// SIMATIC S7-200 project (STEP 7-Micro/WIN), CPU 226 CN REL 02.01

SYMBOL_TABLE USER1
Sens_Tub_Inf     I0.0     // Sensor fotoelectrico del tubo inferior (nivel bajo de stock)
Sens_Tub_Sup     I0.1     // Sensor fotoelectrico del tubo superior (nivel alto de stock)
Sens_Sal_Tub     I0.2     // Sensor de presencia a la salida del tubo dosificador
Sens_Pieza_Rec   I0.3     // Sensor de presencia de pieza lista para recoger
Sens_Fibra_Pza   I0.4     // Sensor de fibra omron (pieza grande receptora presente)
CilS_Ext         I0.5     // Sensor cilindro superior extendido (sujetador OK)
CilS_Ret         I0.6     // Sensor cilindro superior retraido
CilI_Ext         I0.7     // Sensor cilindro inferior extendido
CilI_Ret         I1.0     // Sensor cilindro inferior retraido (pieza liberada)
Giro_AH          I1.1     // Sensor giro antihorario alcanzado (posicion recogida)
Giro_H           I1.2     // Sensor giro horario alcanzado (posicion origen)
Pinza_Cer        I1.3     // Sensor cierre de la pinza de agarre
CilV_Abajo       I1.4     // Sensor cilindro vertical hacia abajo
CilV_Arriba      I1.5     // Sensor cilindro vertical hacia arriba
CilH_Atras       I1.6     // Sensor cilindro horizontal hacia atras (origen)
CilH_Adelante    I1.7     // Sensor cilindro horizontal hacia adelante (sobre pieza)
Btn_Rojo         I2.4     // Boton de parada
Btn_Verde        I2.5     // Boton de marcha
Seta_Emerg       I2.6     // Seta de emergencia (NC - 0 = emergencia activa)
Selector         I2.7     // Selector rotatorio de modo
V_CilI           Q0.0     // Valvula cilindro inferior (liberador) - activa en P2
V_CilS           Q0.1     // Valvula cilindro superior (sujetador) - activa en P1 y P2
V_Giro_H         Q0.2     // Valvula cilindro rotatorio antihorario - activa en P4 a P7
V_Pinza          Q0.3     // Valvula garra (cerrar pinza) - activa en P6 a P9
V_CilV           Q0.4     // Valvula cilindro vertical (bajar) - activa en P5 P6 P9 P10
V_CilH           Q0.5     // Valvula cilindro horizontal (adelante) - activa en P8 a P11
Baliza_Roja      Q0.6     // Baliza roja - sin stock en reposo
Baliza_Amarilla  Q0.7     // Baliza amarilla - parada activa (M6.0)
Baliza_Verde     Q1.0     // Baliza verde - ciclo en ejecucion
Led_Amarillo     Q1.5     // LED boton amarillo - parada activa
Led_Verde        Q1.6     // LED boton verde - ciclo en ejecucion
Led_Rojo         Q1.7     // LED boton rojo - sin stock en reposo
P0_Reposo        M0.0     // Plaza P0 - Estado reposo (marcado inicial)
P1_Dos_Sujetar   M0.1     // Plaza P1 - Cilindro superior sujetando columna
P2_Dos_Caida     M0.2     // Plaza P2 - Cilindro inferior retraido (pieza en caida)
P3_Dos_Restaurar M0.3     // Plaza P3 - Dosificador retornando a posicion base
P4_Mesa_Giro     M0.4     // Plaza P4 - Mesa girando a posicion de recogida
P5_Pick_Bajar    M0.5     // Plaza P5 - Garra descendiendo sobre pieza secundaria
P6_Pick_Agarrar  M0.6     // Plaza P6 - Pinza cerrando para sujetar la pieza
P7_Pick_Subir    M0.7     // Plaza P7 - Garra subiendo con pieza sujeta
P8_Place_Trans   M1.0     // Plaza P8 - Brazo trasladando horizontalmente a base
P9_Place_Bajar   M1.1     // Plaza P9 - Garra bajando para insertar en base
P10_Place_Soltar M1.2     // Plaza P10 - Pinza abriendo para liberar pieza
P11_Place_Subir  M1.3     // Plaza P11 - Garra subiendo tras ensamblaje
P12_Reset_Arm    M1.4     // Plaza P12 - Retorno horizontal y mesa a origen
Ev_Marcha        M2.0     // Evento - Boton de marcha activo
Ev_Tub_Inf       M2.1     // Evento - Stock disponible en tubo (nivel bajo)
Ev_Fibra         M2.2     // Evento - Pieza grande receptora detectada
Ev_CilS_Ext      M2.3     // Evento - Cilindro superior extendido confirmado
Ev_CilS_Ret      M2.4     // Evento - Cilindro superior retraido confirmado
Ev_CilI_Ext      M2.5     // Evento - Cilindro inferior extendido confirmado
Ev_CilI_Ret      M2.6     // Evento - Cilindro inferior retraido (pieza liberada)
Ev_Giro_AH       M2.7     // Evento - Giro antihorario alcanzado (posicion recogida)
Ev_Giro_H        M3.0     // Evento - Giro horario alcanzado (posicion origen)
Ev_Pinza_Cer     M3.1     // Evento - Pinza cerrada (agarre confirmado)
Ev_CilV_Abajo    M3.2     // Evento - Cilindro vertical en posicion abajo
Ev_CilV_Arriba   M3.3     // Evento - Cilindro vertical en posicion arriba
Ev_CilH_Atras    M3.4     // Evento - Cilindro horizontal en posicion atras
Ev_CilH_Adel     M3.5     // Evento - Cilindro horizontal en posicion adelante
T0_Inicio        M4.0     // Disparo T0 - Condicion para iniciar ciclo (P0->P1)
T1_SujecOK       M4.1     // Disparo T1 - Sujecion de columna confirmada (P1->P2)
T2_PiezaCaida    M4.2     // Disparo T2 - Pieza liberada y caida (P2->P3)
T3_DosifRest     M4.3     // Disparo T3 - Dosificador restaurado (P3->P4)
T4_MesaRec       M4.4     // Disparo T4 - Mesa en posicion recogida (P4->P5)
T5_GarraAbajo    M4.5     // Disparo T5 - Garra en contacto con pieza (P5->P6)
T6_AgarreOK      M4.6     // Disparo T6 - Agarre de pieza confirmado (P6->P7)
T7_PiezaElev     M4.7     // Disparo T7 - Pieza secundaria elevada (P7->P8)
T8_BrazoAdel     M5.0     // Disparo T8 - Brazo en punto de entrega (P8->P9)
T9_PiezaBase     M5.1     // Disparo T9 - Pieza posicionada en base grande (P9->P10)
T10_PinzaAb      M5.2     // Disparo T10 - Pinza abierta pieza liberada (P10->P11)
T11_GarraRet     M5.3     // Disparo T11 - Garra retirada del ensamblaje (P11->P12)
T12_FinCiclo     M5.4     // Disparo T12 - Sistema en origen fin de ciclo (P12->P0)
Flag_Parada      M6.0     // Flag de parada - activado por flanco Btn_Rojo reset en P0
Sol_ES           V0.0     // Solicitud Ensamblaje a Seleccion
Ack_Sol_ES       V1.0     // Reconocimiento ES
Ack_ME           V0.1     // Reconocimiento marcha Unidad de Ensamblaje
Marcha_E         V1.1     // Solicitud de marcha para la Unidad de Ensamblaje
Ens_OK           V0.2     // Unidad de Ensamblaje disponible
END_SYMBOL_TABLE

SYMBOL_TABLE S7-200 Symbols
First_Scan_On    SM0.1    // 仅第一个扫描周期中接通为 ON
END_SYMBOL_TABLE

ORGANIZATION_BLOCK MAIN:OB1
TITLE=UNIDAD DE ENSAMBLAJE - RED DE PETRI CIPN v2
//  ===========================================================
//  MODULO 0: SEGURIDAD - EMERGENCIA (Evaluado primero, cada scan)
//  Si Seta = 0 (NC abierta) -> Reset total, fuerza P0, apaga salidas.
//  ===========================================================
BEGIN
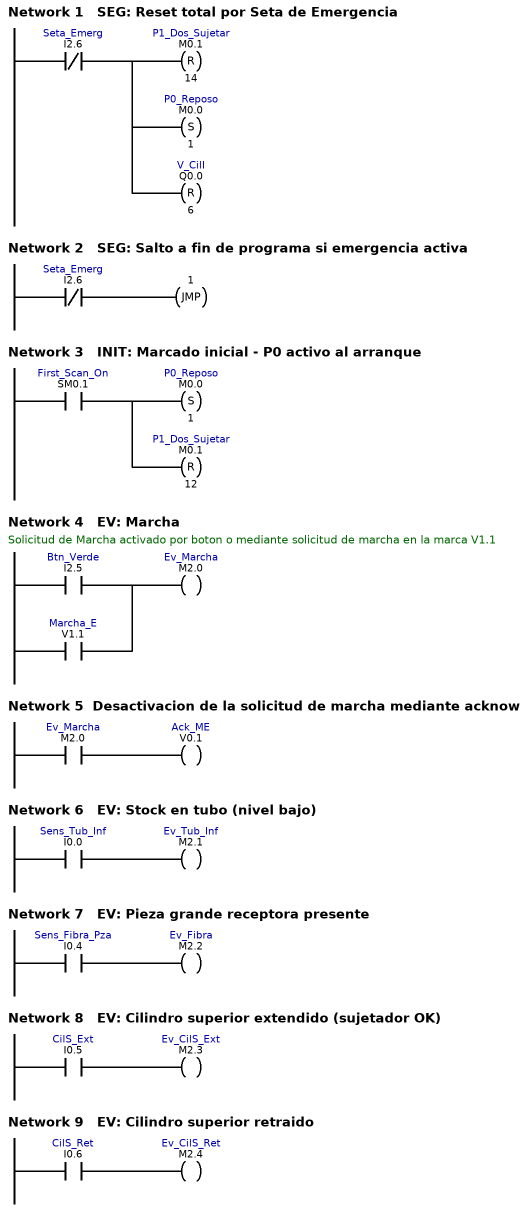
Network 1 //  SEG: Reset total por Seta de Emergencia
LDN    Seta_Emerg:I2.6
R      P1_Dos_Sujetar:M0.1, 14
S      P0_Reposo:M0.0, 1
R      V_CilI:Q0.0, 6
Network 2 //  SEG: Salto a fin de programa si emergencia activa
// ===========================================================
// MODULO 1: INICIALIZACION
// Ejecuta solo en el primer scan (SM0.1 = 1 unicamente en scan 1).
// Establece marcado inicial: P0 activo, resto limpio.
// ===========================================================
LDN    Seta_Emerg:I2.6
JMP    1
Network 3 //  INIT: Marcado inicial - P0 activo al arranque
// ===========================================================
// MODULO 2: EVENTOS (CAPTURA DE SENSORES)
// Copia directa de entradas a marcas de evento para desacoplar
// la logica secuencial de las senales fisicas.
// ===========================================================
LD     First_Scan_On:SM0.1
S      P0_Reposo:M0.0, 1
R      P1_Dos_Sujetar:M0.1, 12
Network 4 //  EV: Marcha 
//  Solicitud de Marcha activado por boton o mediante solicitud de marcha en la marca V1.1
LD     Btn_Verde:I2.5
O      Marcha_E:V1.1
=      Ev_Marcha:M2.0
Network 5 // Desactivacion de la solicitud de marcha mediante acknowledgement
LD     Ev_Marcha:M2.0
=      Ack_ME:V0.1
Network 6 //  EV: Stock en tubo (nivel bajo)
LD     Sens_Tub_Inf:I0.0
=      Ev_Tub_Inf:M2.1
Network 7 //  EV: Pieza grande receptora presente
LD     Sens_Fibra_Pza:I0.4
=      Ev_Fibra:M2.2
Network 8 //  EV: Cilindro superior extendido (sujetador OK)
LD     CilS_Ext:I0.5
=      Ev_CilS_Ext:M2.3
Network 9 //  EV: Cilindro superior retraido
LD     CilS_Ret:I0.6
=      Ev_CilS_Ret:M2.4
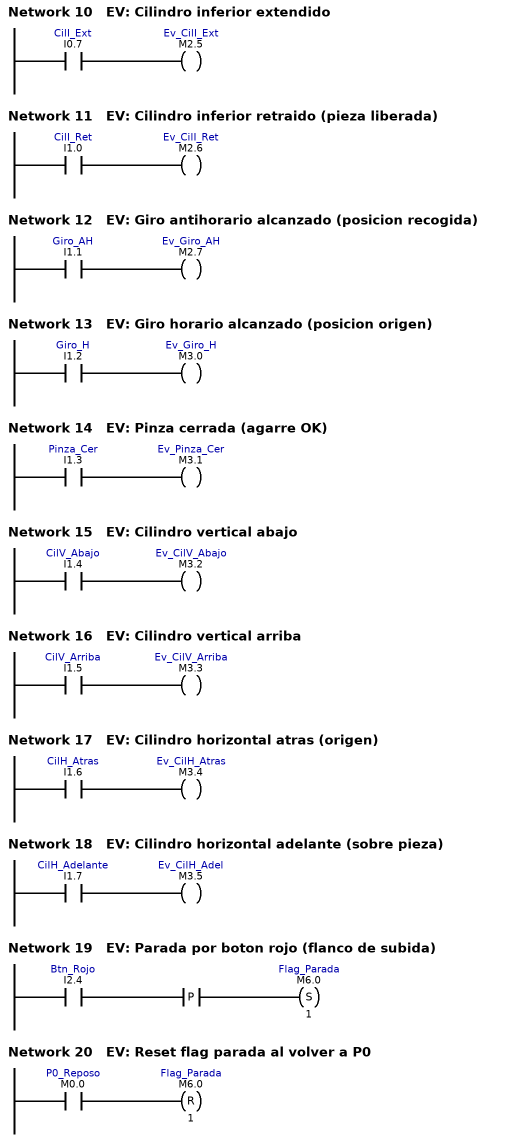
Network 10 //  EV: Cilindro inferior extendido
LD     CilI_Ext:I0.7
=      Ev_CilI_Ext:M2.5
Network 11 //  EV: Cilindro inferior retraido (pieza liberada)
LD     CilI_Ret:I1.0
=      Ev_CilI_Ret:M2.6
Network 12 //  EV: Giro antihorario alcanzado (posicion recogida)
LD     Giro_AH:I1.1
=      Ev_Giro_AH:M2.7
Network 13 //  EV: Giro horario alcanzado (posicion origen)
LD     Giro_H:I1.2
=      Ev_Giro_H:M3.0
Network 14 //  EV: Pinza cerrada (agarre OK)
LD     Pinza_Cer:I1.3
=      Ev_Pinza_Cer:M3.1
Network 15 //  EV: Cilindro vertical abajo
LD     CilV_Abajo:I1.4
=      Ev_CilV_Abajo:M3.2
Network 16 //  EV: Cilindro vertical arriba
LD     CilV_Arriba:I1.5
=      Ev_CilV_Arriba:M3.3
Network 17 //  EV: Cilindro horizontal atras (origen)
LD     CilH_Atras:I1.6
=      Ev_CilH_Atras:M3.4
Network 18 //  EV: Cilindro horizontal adelante (sobre pieza)
LD     CilH_Adelante:I1.7
=      Ev_CilH_Adel:M3.5
Network 19 //  EV: Parada por boton rojo (flanco de subida)
LD     Btn_Rojo:I2.4
EU
S      Flag_Parada:M6.0, 1
Network 20 //  EV: Reset flag parada al volver a P0
// ===========================================================
// MODULO 3: CONDICIONES DE DISPARO (RECEPTIVIDADES)
// Cada transicion Tn se habilita si su plaza de entrada
// tiene marca AND se cumplen las condiciones sensoriales.
// La parada (M6.0) bloquea T0 para no iniciar nuevo ciclo.
// ===========================================================
LD     P0_Reposo:M0.0
R      Flag_Parada:M6.0, 1
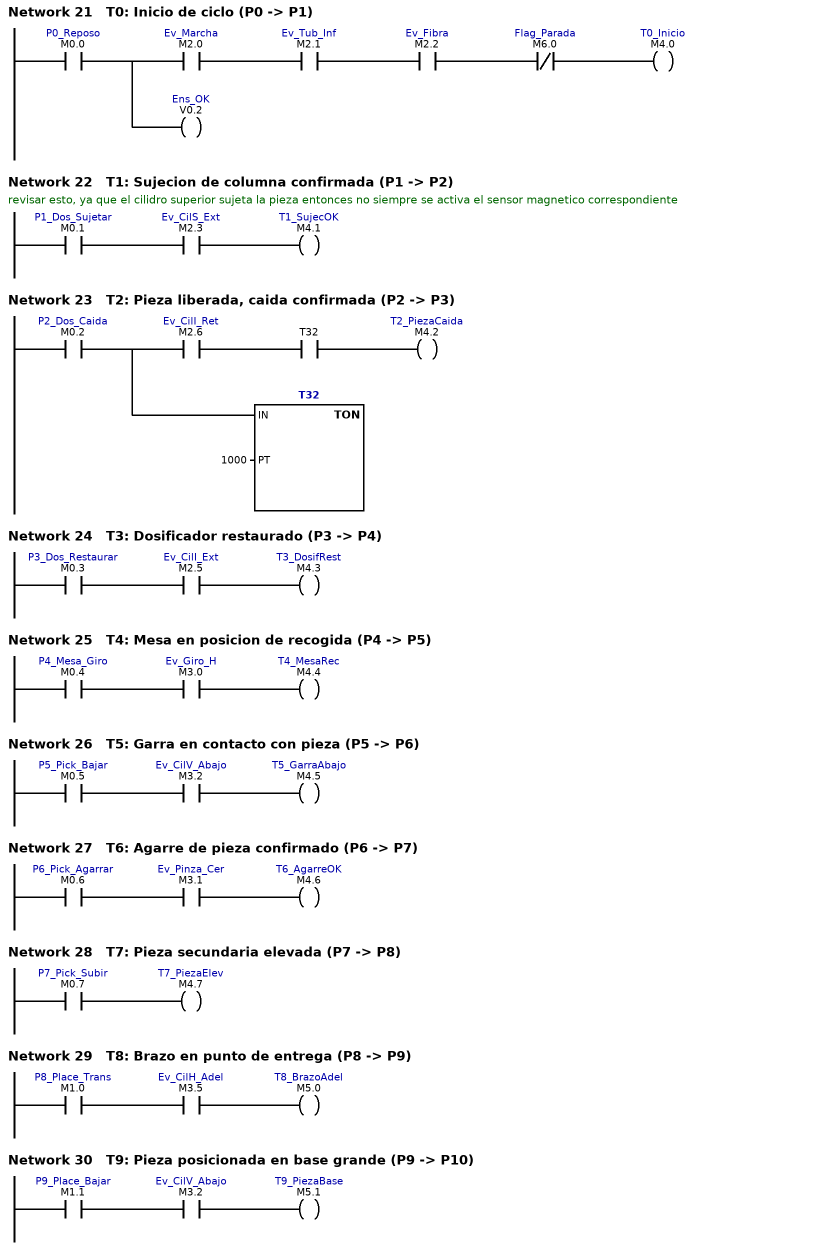
Network 21 //  T0: Inicio de ciclo (P0 -> P1)
LD     P0_Reposo:M0.0
LPS
A      Ev_Marcha:M2.0
A      Ev_Tub_Inf:M2.1
A      Ev_Fibra:M2.2
AN     Flag_Parada:M6.0
=      T0_Inicio:M4.0
LPP
=      Ens_OK:V0.2
Network 22 //  T1: Sujecion de columna confirmada (P1 -> P2)
// revisar esto, ya que el cilidro superior sujeta la pieza entonces no siempre se activa el sensor magnetico correspondiente
LD     P1_Dos_Sujetar:M0.1
A      Ev_CilS_Ext:M2.3
=      T1_SujecOK:M4.1
Network 23 //  T2: Pieza liberada, caida confirmada (P2 -> P3)
LD     P2_Dos_Caida:M0.2
LPS
A      Ev_CilI_Ret:M2.6
A      T32
=      T2_PiezaCaida:M4.2
LPP
TON    T32, 1000
Network 24 //  T3: Dosificador restaurado (P3 -> P4)
LD     P3_Dos_Restaurar:M0.3
A      Ev_CilI_Ext:M2.5
=      T3_DosifRest:M4.3
Network 25 //  T4: Mesa en posicion de recogida (P4 -> P5)
LD     P4_Mesa_Giro:M0.4
A      Ev_Giro_H:M3.0
=      T4_MesaRec:M4.4
Network 26 //  T5: Garra en contacto con pieza (P5 -> P6)
LD     P5_Pick_Bajar:M0.5
A      Ev_CilV_Abajo:M3.2
=      T5_GarraAbajo:M4.5
Network 27 //  T6: Agarre de pieza confirmado (P6 -> P7)
LD     P6_Pick_Agarrar:M0.6
A      Ev_Pinza_Cer:M3.1
=      T6_AgarreOK:M4.6
Network 28 //  T7: Pieza secundaria elevada (P7 -> P8)
LD     P7_Pick_Subir:M0.7
=      T7_PiezaElev:M4.7
Network 29 //  T8: Brazo en punto de entrega (P8 -> P9)
LD     P8_Place_Trans:M1.0
A      Ev_CilH_Adel:M3.5
=      T8_BrazoAdel:M5.0
Network 30 //  T9: Pieza posicionada en base grande (P9 -> P10)
LD     P9_Place_Bajar:M1.1
A      Ev_CilV_Abajo:M3.2
=      T9_PiezaBase:M5.1
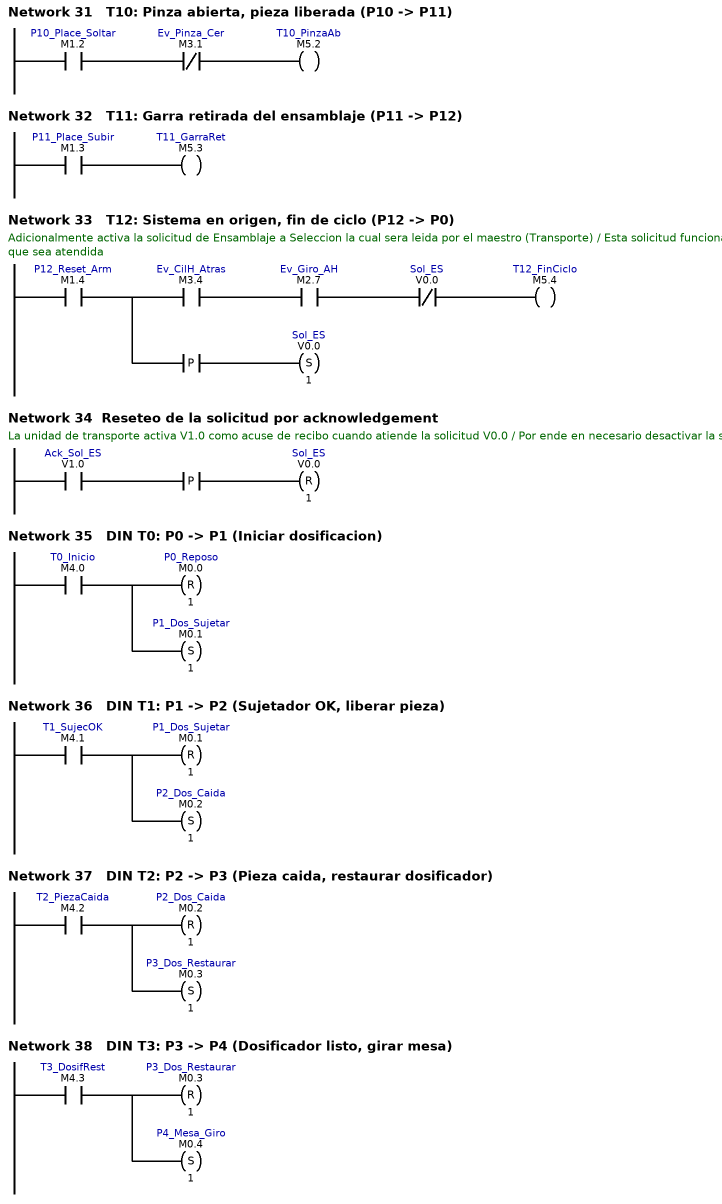
Network 31 //  T10: Pinza abierta, pieza liberada (P10 -> P11)
LD     P10_Place_Soltar:M1.2
AN     Ev_Pinza_Cer:M3.1
=      T10_PinzaAb:M5.2
Network 32 //  T11: Garra retirada del ensamblaje (P11 -> P12)
LD     P11_Place_Subir:M1.3
=      T11_GarraRet:M5.3
Network 33 //  T12: Sistema en origen, fin de ciclo (P12 -> P0)
// Adicionalmente activa la solicitud de Ensamblaje a Seleccion la cual sera leida por el maestro (Transporte)
// Esta solicitud funciona como enclavamiento que impide volver al estado de reposo hasta que sea atendida
// ===========================================================
// MODULO 4: DINAMICA DE LA RED
// Actualiza el marcado. Cada rung corresponde a una transicion.
// SET plaza destino, RESET plaza origen.
// Separados en redes individuales para evitar efecto avalancha.
// ===========================================================
LD     P12_Reset_Arm:M1.4
LPS
A      Ev_CilH_Atras:M3.4
A      Ev_Giro_AH:M2.7
AN     Sol_ES:V0.0
=      T12_FinCiclo:M5.4
LPP
EU
S      Sol_ES:V0.0, 1
Network 34 // Reseteo de la solicitud por acknowledgement
// La unidad de transporte activa V1.0 como acuse de recibo cuando atiende la solicitud V0.0
// Por ende en necesario desactivar la solicitud para evitar repeticiones.
LD     Ack_Sol_ES:V1.0
EU
R      Sol_ES:V0.0, 1
Network 35 //  DIN T0: P0 -> P1 (Iniciar dosificacion)
LD     T0_Inicio:M4.0
R      P0_Reposo:M0.0, 1
S      P1_Dos_Sujetar:M0.1, 1
Network 36 //  DIN T1: P1 -> P2 (Sujetador OK, liberar pieza)
LD     T1_SujecOK:M4.1
R      P1_Dos_Sujetar:M0.1, 1
S      P2_Dos_Caida:M0.2, 1
Network 37 //  DIN T2: P2 -> P3 (Pieza caida, restaurar dosificador)
LD     T2_PiezaCaida:M4.2
R      P2_Dos_Caida:M0.2, 1
S      P3_Dos_Restaurar:M0.3, 1
Network 38 //  DIN T3: P3 -> P4 (Dosificador listo, girar mesa)
LD     T3_DosifRest:M4.3
R      P3_Dos_Restaurar:M0.3, 1
S      P4_Mesa_Giro:M0.4, 1
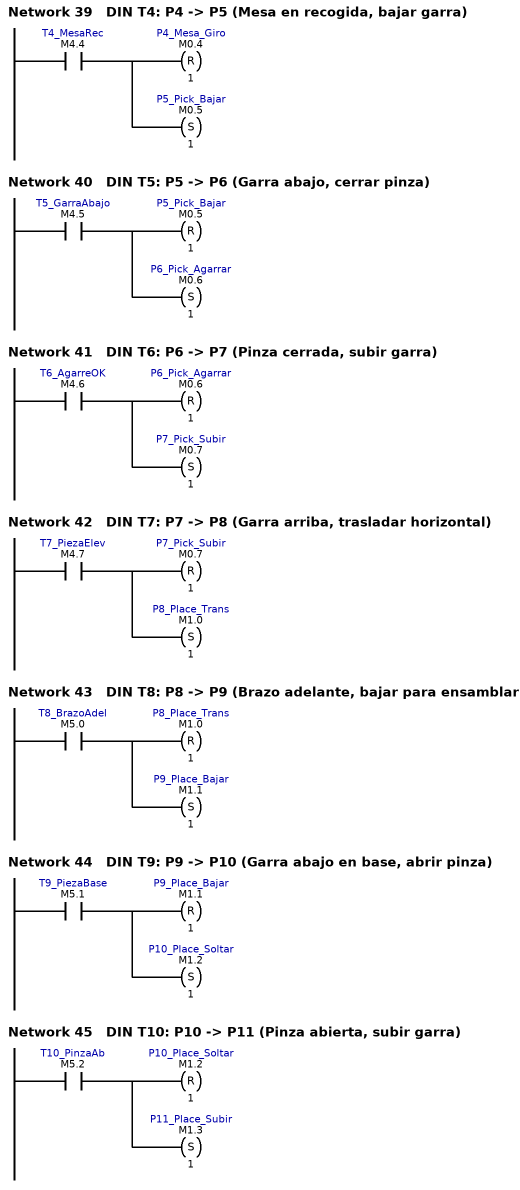
Network 39 //  DIN T4: P4 -> P5 (Mesa en recogida, bajar garra)
LD     T4_MesaRec:M4.4
R      P4_Mesa_Giro:M0.4, 1
S      P5_Pick_Bajar:M0.5, 1
Network 40 //  DIN T5: P5 -> P6 (Garra abajo, cerrar pinza)
LD     T5_GarraAbajo:M4.5
R      P5_Pick_Bajar:M0.5, 1
S      P6_Pick_Agarrar:M0.6, 1
Network 41 //  DIN T6: P6 -> P7 (Pinza cerrada, subir garra)
LD     T6_AgarreOK:M4.6
R      P6_Pick_Agarrar:M0.6, 1
S      P7_Pick_Subir:M0.7, 1
Network 42 //  DIN T7: P7 -> P8 (Garra arriba, trasladar horizontal)
LD     T7_PiezaElev:M4.7
R      P7_Pick_Subir:M0.7, 1
S      P8_Place_Trans:M1.0, 1
Network 43 //  DIN T8: P8 -> P9 (Brazo adelante, bajar para ensamblar)
LD     T8_BrazoAdel:M5.0
R      P8_Place_Trans:M1.0, 1
S      P9_Place_Bajar:M1.1, 1
Network 44 //  DIN T9: P9 -> P10 (Garra abajo en base, abrir pinza)
LD     T9_PiezaBase:M5.1
R      P9_Place_Bajar:M1.1, 1
S      P10_Place_Soltar:M1.2, 1
Network 45 //  DIN T10: P10 -> P11 (Pinza abierta, subir garra)
LD     T10_PinzaAb:M5.2
R      P10_Place_Soltar:M1.2, 1
S      P11_Place_Subir:M1.3, 1
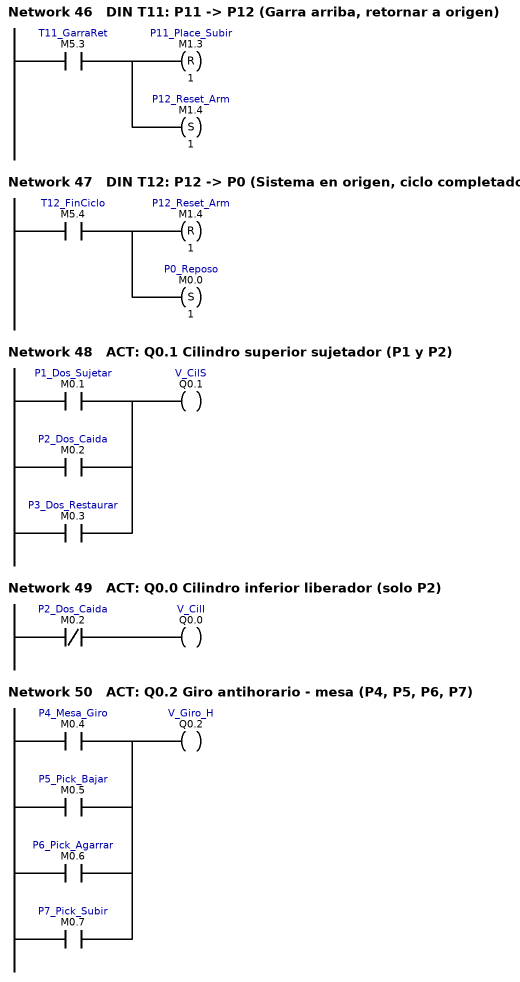
Network 46 //  DIN T11: P11 -> P12 (Garra arriba, retornar a origen)
LD     T11_GarraRet:M5.3
R      P11_Place_Subir:M1.3, 1
S      P12_Reset_Arm:M1.4, 1
Network 47 //  DIN T12: P12 -> P0 (Sistema en origen, ciclo completado)
// ===========================================================
// MODULO 5: ACCIONES (ASIGNACION DE SALIDAS FISICAS)
// Cada salida Q se activa por nivel segun las plazas activas.
// El orden sigue el diseno de la CIPN (3_Diseno_Petri.md).
// Este modulo solo se alcanza si NO hay emergencia activa.
// ===========================================================
LD     T12_FinCiclo:M5.4
R      P12_Reset_Arm:M1.4, 1
S      P0_Reposo:M0.0, 1
Network 48 //  ACT: Q0.1 Cilindro superior sujetador (P1 y P2)
LD     P1_Dos_Sujetar:M0.1
O      P2_Dos_Caida:M0.2
O      P3_Dos_Restaurar:M0.3
=      V_CilS:Q0.1
Network 49 //  ACT: Q0.0 Cilindro inferior liberador (solo P2)
LDN    P2_Dos_Caida:M0.2
=      V_CilI:Q0.0
Network 50 //  ACT: Q0.2 Giro antihorario - mesa (P4, P5, P6, P7)
LD     P4_Mesa_Giro:M0.4
O      P5_Pick_Bajar:M0.5
O      P6_Pick_Agarrar:M0.6
O      P7_Pick_Subir:M0.7
=      V_Giro_H:Q0.2
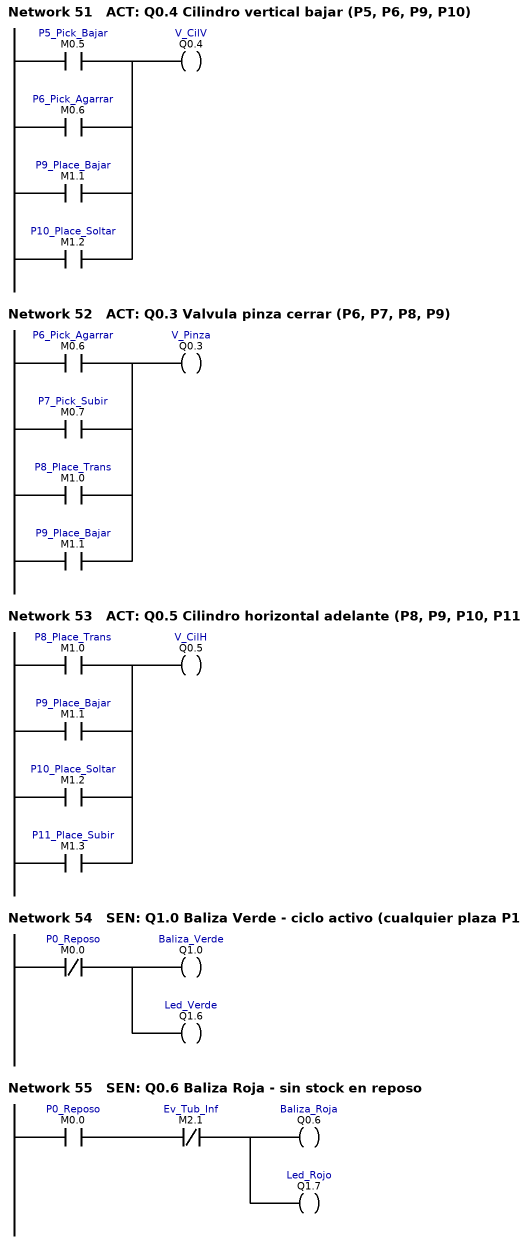
Network 51 //  ACT: Q0.4 Cilindro vertical bajar (P5, P6, P9, P10)
LD     P5_Pick_Bajar:M0.5
O      P6_Pick_Agarrar:M0.6
O      P9_Place_Bajar:M1.1
O      P10_Place_Soltar:M1.2
=      V_CilV:Q0.4
Network 52 //  ACT: Q0.3 Valvula pinza cerrar (P6, P7, P8, P9)
LD     P6_Pick_Agarrar:M0.6
O      P7_Pick_Subir:M0.7
O      P8_Place_Trans:M1.0
O      P9_Place_Bajar:M1.1
=      V_Pinza:Q0.3
Network 53 //  ACT: Q0.5 Cilindro horizontal adelante (P8, P9, P10, P11)
// ===========================================================
// SENALIZACION DE BALIZA Y LEDS
// ===========================================================
LD     P8_Place_Trans:M1.0
O      P9_Place_Bajar:M1.1
O      P10_Place_Soltar:M1.2
O      P11_Place_Subir:M1.3
=      V_CilH:Q0.5
Network 54 //  SEN: Q1.0 Baliza Verde - ciclo activo (cualquier plaza P1-P12)
LDN    P0_Reposo:M0.0
=      Baliza_Verde:Q1.0
=      Led_Verde:Q1.6
Network 55 //  SEN: Q0.6 Baliza Roja - sin stock en reposo
LD     P0_Reposo:M0.0
AN     Ev_Tub_Inf:M2.1
=      Baliza_Roja:Q0.6
=      Led_Rojo:Q1.7
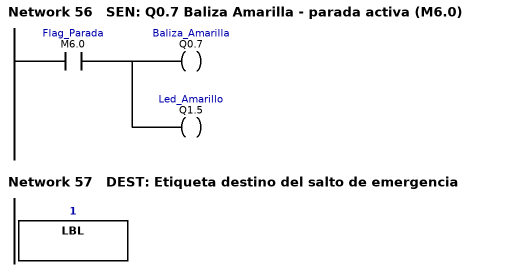
Network 56 //  SEN: Q0.7 Baliza Amarilla - parada activa (M6.0)
// ===========================================================
// DESTINO DEL SALTO DE EMERGENCIA
// LBL 1 debe estar en una red independiente (regla Step7 Micro/WIN)
// ===========================================================
LD     Flag_Parada:M6.0
=      Baliza_Amarilla:Q0.7
=      Led_Amarillo:Q1.5
Network 57 //  DEST: Etiqueta destino del salto de emergencia
LBL    1
END_ORGANIZATION_BLOCK
